// Mitsubishi GX Works2 project: Prática 03 - modbus   PLC: FX3U/FX3UC
// Configuração Modbus RTU

PROGRAM MAIN
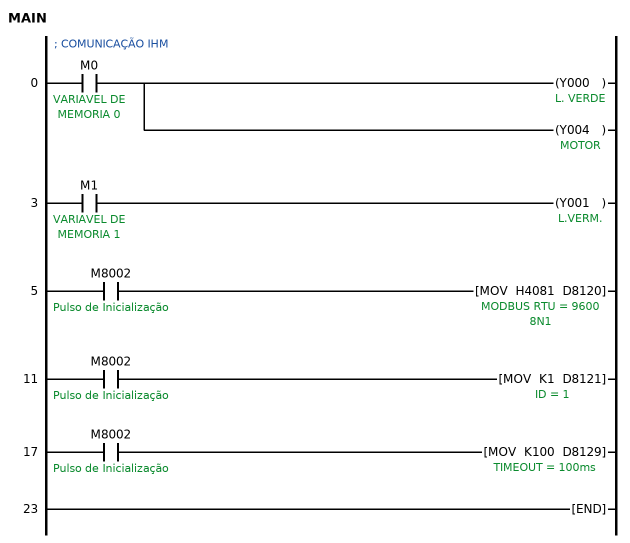
; COMUNICAÇÃO IHM
0     LD      M0  ; VARIAVEL DE MEMORIA 0
      OUT     Y000  ; L. VERDE
      OUT     Y004  ; MOTOR
3     LD      M1  ; VARIAVEL DE MEMORIA 1
      OUT     Y001  ; L.VERM.
5     LD      M8002  ; Pulso de Inicialização
      MOV     H4081 D8120  ; MODBUS RTU = 9600 8N1
11    LD      M8002  ; Pulso de Inicialização
      MOV     K1 D8121  ; ID = 1
17    LD      M8002  ; Pulso de Inicialização
      MOV     K100 D8129  ; TIMEOUT = 100ms
23    END
END_PROGRAM

// device comments not shown above
X000  ; B.LIGAR
X001  ; B. DESLIGAR
Y002  ; RELE 2
Y005  ; SENTIDO
M2  ; VARIAVEL DE MEMORIA 2
M100  ; MEMORIA 100
D0  ; REGISTRO 0
D1  ; SAIDA ANALOGICA
D2  ; ENCHE O TANQUE
D3  ; ESVAZIA O TANQUE
